FUNCTION_BLOCK FB_CleaningMotorAxisCU EXTENDS FB_CleanDevice
VAR_INPUT
  bI_SafeToMove                        : BOOL;
  
  //Limit switches
  bI_ReferenceSensor            AT %I* : BOOL;  (*Physical sensor feedback reference position*)
  
  //Inputs from EL7201 Terminal
  wI_StatusWord                 AT %I* : UINT; (*Status word: 6041:0*)
  lI_EncoderValue               AT %I* : DINT; (*Encoder value*)
  bI_DeviceOnline               AT %I* : BOOL; (*Check link to device*)
  
  fB_Axis                              : FB_EL7201;    //Axis controller
  
  //References
  pC_MsgInterface                      : POINTER TO ST_ADS_MSG_IF;
  iC_BlockId                           : INT;
END_VAR

VAR_OUTPUT
  //Outputs to EL7201 Terminal
  wO_ControlWord                AT %Q* : UINT;                         (*Control word:  6040:0*)
  iO_TargetVelocity             AT %Q* : DINT;                         (*Target velocity:  60FF:0*)
END_VAR

VAR
  //Limit switches
  bL_ReferenceSensor                   : BOOL;  (*Negated sensor feedback reference position*)

  fb_TonDeviceOnline                   : TON;
	bIDp_DeviceReset                     : BOOL := FALSE;
	fb_RTrigDeviceReset                  : R_TRIG;

  bL_SafeRunningCondition              : BOOL;
  bL_SafeMoveNeg                       : BOOL;
  bL_SafeMovePos                       : BOOL;
  bL_memRefSensor                      : BOOL;
  bL_FirstRun                          : BOOL := TRUE;

  fL_ManualMoveTolerance               : REAL := 0.001;
  
  bL_InPosCappClean                    : BOOL;
  bL_InPosPark                         : BOOL;
  
  wL_ErrorCode                         : WORD;
  
  (*Messaging*)
  fB_MsgQueue                          : FB_MSG_QUEUE;
  fB_MsgHandler                        : FB_MSG_HANDLER;
  sL_MsgConfig                         : ST_MSG_CONFIG;
  fB_Msg                               : ARRAY [1..iC_NUM_MSG] OF FB_MESSAGE;
END_VAR

VAR PERSISTENT
  fI_PositionCappingClean              : REAL;           (*[mm]*)
  fI_PositionPark                      : REAL;           (*[mm]*)
  fI_PositionTolerance                 : REAL := 0.001;  (*[m]*)
  sI_SpeedDef                          : ST_SPEEDS;  (*Speed defs [mm/s]*)
END_VAR

VAR CONSTANT
  iC_NUM_MSG                           : INT  := 1;
END_VAR

//Limit switches for internal use
bL_ReferenceSensor := NOT bI_ReferenceSensor;

(*----------------------------------------------------------------------------------------------------------------------------------------------- *)
(*Running Conditions for Cleaning Unit  *)
(*----------------------------------------------------------------------------------------------------------------------------------------------- *)
IF I_MachineStatus.pSafetyOk AND I_MachineStatus.pMachineReady AND (wL_ErrorCode = 0 OR wL_ErrorCode.5)THEN  (*Dont check limit switch here*)
  bL_SafeRunningCondition := TRUE;
ELSE
  bL_SafeRunningCondition := FALSE;
END_IF;

bL_SafeMoveNeg := bL_SafeRunningCondition AND NOT bL_ReferenceSensor AND bI_SafeToMove;
bL_SafeMovePos := bL_SafeRunningCondition AND bI_SafeToMove;

(*Because the WcState sets an error for on cycle, we use this timer to check if the bus is down.*)
fb_TonDeviceOnline(IN := bI_DeviceOnline, PT := T#20MS);
fb_RTrigDeviceReset(CLK := bIDp_DeviceReset);
IF fb_TonDeviceOnline.Q OR fb_RTrigDeviceReset.Q THEN
  bL_RefKnown    := FALSE;        (*Reset Reference when link to device is lost, e.g. when machine power off*)
	wL_ErrorCode.9 := TRUE;
END_IF;

(*----------------------------------------------------------------------------------------------------------------------------------------------- *)
(*Position detection*)
(*----------------------------------------------------------------------------------------------------------------------------------------------- *)
IF     fB_Axis.fO_ActualPosition >= ((fI_PositionCappingClean / 1000) - fI_PositionTolerance)
   AND fB_Axis.fO_ActualPosition <= ((fI_PositionCappingClean / 1000) + fI_PositionTolerance)
THEN
  bL_InPosCappClean := TRUE;
  bL_InPosPark      := FALSE;
ELSIF  fB_Axis.fO_ActualPosition >= ((fI_PositionPark / 1000) - fI_PositionTolerance)
   AND fB_Axis.fO_ActualPosition <= ((fI_PositionPark / 1000) + fI_PositionTolerance)
THEN
  bL_InPosCappClean := FALSE;
  bL_InPosPark      := TRUE;
ELSE
  bL_InPosCappClean := FALSE;
  bL_InPosPark      := FALSE;
END_IF;


(*----------------------------------------------------------------------------------------------------------------------------------------------- *)
(* Axis control  *)
(*----------------------------------------------------------------------------------------------------------------------------------------------- *)
fB_Axis.bI_RegActive := bL_SafeRunningCondition AND NOT bL_Error; //Activate controller
fB_Axis.bI_EStop     := I_MachineStatus.pSafetyOk;                //negative logic for bI_EStop

fB_Axis(wI_StatusWord := wI_StatusWord ,lI_EncoderValue := lI_EncoderValue);

fB_Axis.bI_FaultReset := FALSE;

wO_ControlWord    := fB_Axis.wO_ControlWord;
iO_TargetVelocity := fB_Axis.iO_TargetVelocity;


(*----------------------------------------------------------------------------------------------------------------------------------------------- *)
(* Supervision  *)
(*----------------------------------------------------------------------------------------------------------------------------------------------- *)
(*
TODO: Supervisor
tL_TimerSurv.PT := T#3S;
tL_TimerSurv();
tL_TimerSensor.PT := T#105s  ;  (* 1meter at 10mm*)
tL_TimerSensor();*)

IF bL_FirstRun THEN
  bL_FirstRun     := FALSE;
  bL_memRefSensor := bL_ReferenceSensor;
END_IF;

(*----------------------------------------------------------------------------------------------------------------------- *)
(*--------------------------------- Fault Diagnosis and Management  ----------------------------------------------------- *)
(*----------------------------------------------------------------------------------------------------------------------- *)
mErrorHandling();

(*----------------------------------------------------------------------------------------------------------------------- *)
(* Messaging                                                                                                              *)
(*----------------------------------------------------------------------------------------------------------------------- *)
fB_MsgHandler();
fB_Msg[1](bI_Status := bL_Error);
fB_MsgQueue();

METHOD mAckError 
VAR_INPUT
END_VAR
wL_ErrorCode := 0;
mErrorHandling();
fB_Axis.bI_FaultReset := TRUE;
END_METHOD

METHOD mCapping : BOOL
VAR_INPUT
  iI_Step    : INT;
  bI_ExitCap : BOOL;
END_VAR
//Abort: Stop whereever axis is and return
IF bL_AbortReq THEN
  fB_Axis.bI_MoveEnable := FALSE;
  bL_Busy  := FALSE;
  bL_Ready := TRUE;

  RETURN;
END_IF

//Normal operation
bL_Ready := FALSE;
CASE iI_Step OF
	0: //Init - Check if axis is not activated, restore safety
    fB_Axis.bI_MoveEnable := FALSE;
		bL_Busy := FALSE;

  1: //Wait for PU axis to lift
    fB_Axis.bI_MoveEnable   := FALSE;
    bL_Busy                 := FALSE;
    
  2: //Wait for CU axis to move in
    mAckError();
    fB_Axis.fI_TargetPosition := (fI_PositionCappingClean / 1000);
    fB_Axis.fI_SpeedLimit     := sI_SpeedDef.fP_PlaceSpeed / 1000;
    
    IF bL_InPosCappClean THEN
      fB_Axis.bI_MoveEnable := FALSE;
      bL_Busy               := FALSE;
      bL_Ready              := TRUE;  //Operation complete
    ELSE
      fB_Axis.bI_MoveEnable := bL_SafeMovePos;
      bL_Busy               := TRUE;
    END_IF
    
  3: //Move CH to park positiom 
    fB_Axis.bI_MoveEnable   := FALSE;
    bL_Busy                 := FALSE;
    
  4: //Wait for PU axis to lower
    fB_Axis.bI_MoveEnable   := FALSE;
    bL_Busy                 := FALSE;
    
	5: //End - Do nothing, capping process active
    mAckError();
		bL_Busy  := FALSE;
    bL_Ready := TRUE;  //Operation complete

	ELSE
		bL_Busy  := FALSE;		
    bL_Ready := TRUE;  //Operation complete
END_CASE
END_METHOD

METHOD mCleaning : BOOL
VAR_INPUT
  iI_Step : INT;
END_VAR
//Abort: Stop whereever axis is and return
IF bL_AbortReq THEN
  fB_Axis.bI_MoveEnable := FALSE;
  bL_Busy  := FALSE;
  bL_Ready := TRUE;

  RETURN;
END_IF

//Normal operation
bL_Ready := FALSE;
CASE iI_Step OF
  0: //Init - Check if axis is not activated, restore safety
    bL_Busy := FALSE;

  1: //Wait for PU axis to lift
    fB_Axis.bI_MoveEnable   := FALSE;
    bL_Busy                 := FALSE;
    
  2: //Wait for CU axis to move in
    mAckError();
    fB_Axis.fI_TargetPosition := (fI_PositionCappingClean / 1000);
    fB_Axis.fI_SpeedLimit     := sI_SpeedDef.fP_PlaceSpeed / 1000;
    
    IF bL_InPosCappClean THEN
      fB_Axis.bI_MoveEnable := FALSE;
      bL_Busy               := FALSE;
      bL_Ready              := TRUE;  //Operation complete
    ELSE
      fB_Axis.bI_MoveEnable := bL_SafeMovePos;
      bL_Busy               := TRUE;
    END_IF
    
  3: //Wait for PU axis to lower
    fB_Axis.bI_MoveEnable   := FALSE;
    bL_Busy                 := FALSE;
    
  4: //Ensure CH axis is at starting position
    fB_Axis.bI_MoveEnable   := FALSE;
    bL_Busy                 := FALSE;
    
  5: //Move CH to clean start position
    fB_Axis.bI_MoveEnable   := FALSE;
    bL_Busy                 := FALSE;

  6: //Wait until cleaning equipment ready
    fB_Axis.bI_MoveEnable   := FALSE;
    bL_Busy                 := FALSE;
    
  7: //Cleaning
    fB_Axis.bI_MoveEnable   := FALSE;
    bL_Busy                 := FALSE;  
    
  8: //Wait until cleaning equipment ready
    fB_Axis.bI_MoveEnable   := FALSE;
    bL_Busy                 := FALSE;
    
  9: //Move CH to end position
    fB_Axis.bI_MoveEnable   := FALSE;
    bL_Busy                 := FALSE;  
    
  10: //Wait for PU axis to lift
    fB_Axis.bI_MoveEnable   := FALSE;
    bL_Busy                 := FALSE;  
  
  11: //Move CH back to start 
    fB_Axis.bI_MoveEnable   := FALSE;
    bL_Busy                 := FALSE;  

  12: //Wait for PU axis to lower
    fB_Axis.bI_MoveEnable   := FALSE;
    bL_Busy                 := FALSE;
    
  13: //End
    fB_Axis.bI_MoveEnable   := FALSE;
    bL_Busy                 := FALSE;  
    bL_Ready                := TRUE;  //Operation complete

  ELSE
    bL_Busy  := FALSE;    
    bL_Ready := TRUE;  //Operation complete
END_CASE
END_METHOD

METHOD PRIVATE mErrorHandling
VAR_INPUT
END_VAR
fB_Msg[1].bI_Status := FALSE;

IF (sI_SpeedDef.fP_PlaceSpeed = 0) OR (sI_SpeedDef.fP_WorkSpeed = 0) OR (sI_SpeedDef.fP_ServiceSpeed = 0) THEN	(* Speed Configuration not done *)
	wL_ErrorCode.6 := TRUE;
END_IF;

IF (fI_PositionCappingClean = 0) THEN		(* Position Configuration not done *)
	wL_ErrorCode.7 := TRUE;
END_IF;

IF fB_Axis.eO_EL7201Status = eFault  THEN
	wL_ErrorCode.8 := TRUE;						(* EL7342 module fault *)
	fB_Msg[1].bI_Status := TRUE;
END_IF;


IF wl_ErrorCode = 0 THEN
	bL_Error := FALSE;
ELSE
	bL_Error := TRUE;
END_IF;
END_METHOD

METHOD mErrorRecovery : BOOL
VAR_INPUT
    iI_Step : INT;
END_VAR
//Do nothing
bL_Busy  := FALSE;
bL_Ready := TRUE;
END_METHOD

METHOD mInit
VAR_INPUT
END_VAR
(*Messages*)
sL_MsgConfig.bI_Enable       := TRUE;
sL_MsgConfig.pI_FbMsgHandler := ADR(fB_MsgHandler);
fB_MsgHandler.pI_MsgQueue    := ADR(fB_MsgQueue);
fB_MsgQueue.pI_MsgInterface  := pC_MsgInterface;
fB_MsgQueue.cI_MaxElement    := 5;

fB_Msg[1].iI_MsgLocation     := iC_BlockId;
fB_Msg[1].pI_MsgConfig       := ADR(sL_MsgConfig);
fB_Msg[1].iI_MsgNumber       := eCMa_AxisErrorX;
END_METHOD

METHOD mManuellMove : BOOL
VAR_INPUT
  bI_Do                  : BOOL;
  fI_TargetPosition      : REAL;
  fL_ManualMoveTolerance : REAL;
END_VAR
fB_Axis.fI_SpeedLimit     := sI_SpeedDef.fP_ServiceSpeed / 1000;
fB_Axis.fI_TargetPosition := fI_TargetPosition / 1000;
IF fB_Axis.fI_TargetPosition > fB_Axis.fO_ActualPosition THEN
  fB_Axis.bI_MoveEnable   := bI_Do AND bL_SafeMovePos;
ELSIF fB_Axis.fI_TargetPosition < fB_Axis.fO_ActualPosition THEN
  fB_Axis.bI_MoveEnable   := bI_Do AND bL_SafeMoveNeg;
ELSE
  fB_Axis.bI_MoveEnable   := bI_Do;
END_IF

bL_Busy  := ABS(fB_Axis.fI_TargetPosition - fB_Axis.fO_ActualPosition) > fL_ManualMoveTolerance;
bL_Ready := NOT (ABS(fB_Axis.fI_TargetPosition - fB_Axis.fO_ActualPosition) > fL_ManualMoveTolerance);  //Operation complete
END_METHOD

METHOD mProduction : BOOL
VAR_INPUT
  iI_Step : INT;
END_VAR
//Abort: Stop whereever axis is and return
IF bL_AbortReq THEN
  fB_Axis.bI_MoveEnable := FALSE;
  bL_Busy  := FALSE;
  bL_Ready := TRUE;

  RETURN;
END_IF

//Normal operation
bL_Ready := FALSE;
CASE iI_Step OF
  0: //Init - Check if axis is not activated, restore safety
    bL_Busy := FALSE;

  1: //Wait for PU axis to lift
    fB_Axis.bI_MoveEnable   := FALSE;
    bL_Busy                 := FALSE;
    
  2: //Wait for CU axis to move out
    mAckError();
    fB_Axis.fI_TargetPosition := (fI_PositionPark / 1000);
    fB_Axis.fI_SpeedLimit     := sI_SpeedDef.fP_PlaceSpeed / 1000;
    
    IF bL_InPosPark THEN
      fB_Axis.bI_MoveEnable := FALSE;
      bL_Busy               := FALSE;
      bL_Ready              := TRUE;  //Operation complete
    ELSE
      fB_Axis.bI_MoveEnable := bL_SafeMoveNeg;
      bL_Busy               := TRUE;
    END_IF
    
  3: //Wait for PU axis to lower
    fB_Axis.bI_MoveEnable   := FALSE;
    bL_Busy                 := FALSE;
    
  4: //End
    fB_Axis.bI_MoveEnable := FALSE;
    bL_Busy               := FALSE;  
    bL_Ready              := TRUE;  //Operation complete

  ELSE
    bL_Busy  := FALSE;    
    bL_Ready := TRUE;  //Operation complete
END_CASE
END_METHOD

METHOD mService : BOOL
VAR_INPUT
  iI_Step : INT;
END_VAR
//Abort: Stop whereever axis is and return
IF bL_AbortReq THEN
  fB_Axis.bI_MoveEnable := FALSE;
  bL_Busy  := FALSE;
  bL_Ready := TRUE;

  RETURN;
END_IF

//Normal operation
bL_Ready := FALSE;
CASE iI_Step OF
  0: //Init - Check if axis is not activated, restore safety
    bL_Busy := FALSE;

  1: //Wait for PU axis to lift to ExitCapping
    fB_Axis.bI_MoveEnable   := FALSE;
    bL_Busy                 := FALSE;
    
  2: //Wait for CU axis to move in
    mAckError();
    fB_Axis.fI_TargetPosition := (fI_PositionPark / 1000);
    fB_Axis.fI_SpeedLimit     := sI_SpeedDef.fP_PlaceSpeed / 1000;
    
    IF bL_InPosPark THEN
      fB_Axis.bI_MoveEnable := FALSE;
      bL_Busy               := FALSE;
      bL_Ready              := TRUE;  //Operation complete
    ELSE
      fB_Axis.bI_MoveEnable := bL_SafeMoveNeg;
      bL_Busy               := TRUE;
    END_IF
    
  3: //End
    fB_Axis.bI_MoveEnable := FALSE;
    bL_Busy               := FALSE;  
    bL_Ready              := TRUE;

  ELSE
    bL_Busy  := FALSE;    
    bL_Ready := TRUE;  //Operation complete
END_CASE
END_METHOD

METHOD mStartup : BOOL
VAR_INPUT
  iI_Step : INT;
END_VAR
CASE iI_Step OF
	0: //Init - Check if axis is not activated, restore safety
		bL_Busy := FALSE;

	1: //Wait until other axes in place
		bL_Busy := FALSE;

	2: //Begin - Init CU axis if NOT bL_RefKnown
    bL_Busy  := NOT bL_RefKnown;
    bL_Ready := bL_RefKnown;
    
    fB_Axis.bI_SetPosition := bL_RefKnown;
    
    IF NOT bL_RefKnown THEN  (* if the CU axis hasn't been initialized with Ref Sensor*)
      IF bL_ReferenceSensor AND NOT bL_memRefSensor AND NOT bL_RefKnown THEN
        bL_RefKnown             := TRUE;                      (* When the sensor is activated, Save the correction value*)
        fB_Axis.bI_SetPosition  := TRUE;                      (*Initialize position to preset value*)
        fB_Axis.bI_MoveEnable   := FALSE;
        bL_Ready                := TRUE;
      ELSE
        IF bL_ReferenceSensor AND bL_memRefSensor THEN
          fB_Axis.fI_TargetPosition := fB_Axis.fO_ActualPosition + 0.01;  (*@@@@CONST, change to JOG_NEGATIVE*)
          fB_Axis.fI_SpeedLimit     := sI_SpeedDef.fP_ServiceSpeed / 1000;     (* Start backward motion, the motor will run until Ref Sensor is ON*)
          fB_Axis.bI_MoveEnable     := bL_SafeMovePos;
        ELSE
          fB_Axis.fI_TargetPosition := -100.0;                               (*@@@@CONST, change to JOG_NEGATIVE*)
          fB_Axis.fI_SpeedLimit     := sI_SpeedDef.fP_ServiceSpeed / 1000;  (* Start backward motion, the motor will run until Ref Sensor is ON*)
          fB_Axis.bI_MoveEnable     := bL_SafeMoveNeg;
        END_IF;
      END_IF;
    END_IF;

    bL_memRefSensor := bL_ReferenceSensor;				(* Memorization of the Ref sensor state for edge detection*)

	3,4: //End
		bL_Busy  := FALSE;		
    bL_Ready := TRUE;  //Operation complete

	ELSE
		bL_Busy  := FALSE;		
    bL_Ready := TRUE;  //Operation complete
END_CASE
END_METHOD

{attribute 'monitoring' := 'call'}
PROPERTY pInPosCappingClean : BOOL
GET
pInPosCappingClean := bL_InPosCappClean;
END_GET
END_PROPERTY

{attribute 'monitoring' := 'call'}
PROPERTY pInPosPark : bool
GET
pInPosPark := bL_InPosPark;
END_GET
END_PROPERTY

END_FUNCTION_BLOCK

(* stored: Version 1.1.0.1, ProductVersion 3.1.4024.9
   POU FB_CleaningMotorAxisCU: Id {412578c3-cbc3-4477-b022-cff4142d0a7e}, SpecialFunc None
   Method mAckError: Id {407264f4-784c-4956-be85-a1db324c160a}
   Method mCapping: Id {f7d65b00-bbb1-446b-89ca-e1dd2bfffb27}
   Method mCleaning: Id {691e3143-62bb-4da6-b284-88163dc74e39}
   Method mErrorHandling: Id {279c74e6-e699-4d87-b088-f07f5c886c73}
   Method mErrorRecovery: Id {17f9780d-a9b8-471b-ba1a-d433341f3aea}
   Method mInit: Id {30b2322a-e2a6-45bb-84a7-a1fd0aad5edb}
   Method mManuellMove: Id {106f9cc4-9aab-4f85-ae8e-947eeea9ca13}
   Method mProduction: Id {fb024e55-d8da-428b-9cbb-78a28f0c9c0d}
   Method mService: Id {4f7a55d6-c286-44f7-b12f-d50a50aae8c5}
   Method mStartup: Id {991de41f-c9c0-49b0-b6df-4461f8e7bfb3}
   Property pInPosCappingClean: Id {c136ee31-7284-4653-9db8-afa62ad84b73}
   Get Get: Id {bc785218-415c-4619-99b2-f19007b13cbe}
   Property pInPosPark: Id {f42bbb15-74a2-4396-8085-65fc9f9552dd}
   Get Get: Id {02be8511-6c6a-4d2b-a906-0c7fcfb04523} *)
